VAR_GLOBAL
	stGroupRef			: AXES_GROUP_REF;
	stAxis				: ARRAY[1..cAxesCount] OF AXIS_REF;
END_VAR

VAR_GLOBAL CONSTANT
	cAxesCount			: UINT:=4;
END_VAR

(* stored: Version 1.1.0.1, ProductVersion 3.1.0.38
   GVL GVL: Id {0de60e34-0e2d-4b10-b51a-624a60cec6ea} *)
